{attribute 'qualified_only'}
{attribute 'strict'}
TYPE StationSequence :
(
	Idle,
	MoverPresent,
	RobotActive,
	DischargeMover,
	Error		
);
END_TYPE

(* stored: Version 1.1.0.1, ProductVersion 3.1.4026.8
   DUT StationSequence: Id {1902de7b-9844-06dc-0f39-280193ecc01b} *)
